Staubli VAL3: onSpaceEvent.pgx

program onSpaceEvent(bool& x_bSave[])
begin
  // edit the action related to the point
  call editAction(x_bSave)
  nSelect=nIndex
  // refresh all
  use:bUseRefresh=true
end
